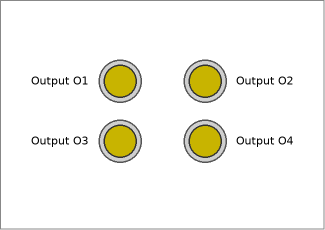
VISUALIZATION V_DO  // 325x230
    Lamp1 (95,56 50x50), variable: HMI_IO.bDOStartLamp, style: Lamp-Lamp1-Yellow
    Lamp1 (180,56 50x50), variable: HMI_IO.bMCForwardlamp, style: Lamp-Lamp1-Yellow
    Lamp1 (95,116 50x50), variable: HMI_IO.bDOResetLamp, style: Lamp-Lamp1-Yellow
    Lamp1 (180,116 50x50), variable: HMI_IO.bDOReverselamp, style: Lamp-Lamp1-Yellow
    Label (25,66 70x30), "Output O1"
    Label (25,126 70x30), "Output O3"
    Label (230,66 70x30), "Output O2"
    Label (230,126 70x30), "Output O4"
END_VISUALIZATION

(* stored: Version 1.1.0.1, ProductVersion 3.1.4024.11
   Visu V_DO: Id {d105f602-051c-4f31-94ad-417b54fa45aa} *)
